(* CODESYS project Project1.project

Project tree, tasks and I/O mapping:
  PLC_AC500_V3 : PM5650-2ETH, ABB Automation Products GmbH, order no. 1SAPx41000R0278, version 3.4.1.0
    application Application
      task Task (cyclic, interval t#10ms, priority 15, watchdog t#20ms x 1) calls PLC_PRG
      CheckConfigurationObject
      program PLC_PRG [ST]
      data type motorIn
      data type motorOut
      data type fanIn
      data type fanOut
      data type valveIn
      data type valveOut
      function block AnalogSensor [ST]
      function block Valve [ST]: close, open, error
      function block AnalogValve [ST]
      function block Motor [ST]: start, stop, error, Init
      interface ILogging: Imethod1, Imethod2
      function block AbsLogging [ST]: Method1
      function block Compressor [ST]
      function block Condensor [ST]
      function block Evaporator [ST]
      function block Fan [ST]
      function block Pressure [ST]: Prop1, Prop2
      function block Temperature [ST]: HiAlarm, LoAlarm
      Diagnosis/
        text list Diag_IO_Bus
        text list Diag_V3_PLC
    IO_Bus : I/O-Bus, ABB Automation Products GmbH, version 3.4.0.0
    Interfaces : Interfaces, ABB Automation Products GmbH, version 3.4.1.0
      COM
      CAN
      Ethernet : Ethernet, ABB Automation Products GmbH, version 3.4.1.0
        ETH1 : IP Settings, ABB Automation Products GmbH, version 3.4.1.0
          NetConfig : NetConfig, ABB Automation Products GmbH, version 3.4.0.0
        ETH2 : IP Settings, ABB Automation Products GmbH, version 3.4.1.0
          NetConfig_1 : NetConfig, ABB Automation Products GmbH, version 3.4.0.0
        Protocols : Client Protocols, ABB Automation Products GmbH, version 3.4.1.0
    Extension_Bus : Extension Bus, ABB Automation Products GmbH, version 3.4.0.0
      Slot_1
      Slot_2
  Panel_CP600 : CP600 Control Panel, ABB Automation Products GmbH, order no. 1SAP500900R0001, version 2.10.0.0
    Panel Project
  libraries: VisuSymbols, 3.5.10.0 (System)
  text list GlobalTextList
*)

// PLC_AC500_V3/Application/motorIn
TYPE motorIn :
STRUCT
	StartMotor:BOOL;
	StopMotor:BOOL;
	Running:BOOL;
	Simulation:BOOL;
END_STRUCT
END_TYPE

// PLC_AC500_V3/Application/motorOut
TYPE motorOut :
STRUCT
	Output:BOOL;
	Error:BOOL;
END_STRUCT
END_TYPE

// PLC_AC500_V3/Application/fanIn
TYPE fanIn EXTENDS motorIn :
STRUCT
	fanSpeed:REAL;
END_STRUCT
END_TYPE

// PLC_AC500_V3/Application/fanOut
TYPE fanOut EXTENDS motorOut :
STRUCT
	outSpeed:REAL;
END_STRUCT
END_TYPE

// PLC_AC500_V3/Application/valveIn
TYPE valveIn :
STRUCT
	OpenCmd:BOOL;
	CloseCmd:BOOL;
	Opened:BOOL;
	Closed:BOOL;
END_STRUCT
END_TYPE

// PLC_AC500_V3/Application/valveOut
TYPE valveOut :
STRUCT
	Output:BOOL;
	Stall:BOOL;
END_STRUCT
END_TYPE

// PLC_AC500_V3/Application/AbsLogging/AMethod1
METHOD PUBLIC ABSTRACT AMethod1 : BOOL
VAR_INPUT
END_VAR

// PLC_AC500_V3/Application/AbsLogging/AMethod2
METHOD PUBLIC ABSTRACT AMethod2 : BOOL
VAR_INPUT
END_VAR

// PLC_AC500_V3/Application/PLC_PRG
PROGRAM PLC_PRG
VAR
	Compressor1:Compressor;
	Evaporator1:Evaporator;
	Condensor1:Condensor;
	
	TT1:Temperature; // Compressor Inlet Temperature / Evaporator Outlet Temperature
	TT2:Temperature; // Compressor Outlet Temperature / Condensor Inlet Temperature
	TT3:Temperature; // Condensor Outlet Temperature / Evaporator Inlet Temperature
	
	PT1:Pressure; // Compressor Inlet Pressure / Evaporator Outlet Pressure
	PT2:Pressure; // Compressor Outlet Pressure / Condensor Inlet Pressure
	PT3:Pressure; // Condensor Outlet Pressure / Evaporator Inlet Pressure
	PT4:Pressure; // 
	
	EEV1:AnalogValve; // Temperature Controlling Valve

	defrostTemperature:REAL;
	chillTemperature:REAL;
	Defrost:BOOL;
	Chilling:BOOL;
	
	var1:REAL;
END_VAR

Compressor1();
Condensor1();
Evaporator1();
PT1();
PT2();
PT3();
PT4();
TT1();
TT2();
TT3();
EEV1();
TT1.EngMax:=100;
TT1.EngMin:=0;
TT1.RawMax:=20000;
TT1.RawMin:=0;
TT1.Simulation:=TRUE;

TT2.EngMax:=100;
TT2.EngMin:=0;
TT2.RawMax:=20000;
TT2.RawMin:=0;
TT2.Simulation:=TRUE;

TT3.EngMax:=100;
TT3.EngMin:=0;
TT3.RawMax:=20000;
TT3.RawMin:=0;
TT3.Simulation:=TRUE;

PT1.EngMax:=10;
PT1.EngMin:=0;
PT1.RawMax:=20000;
PT1.RawMin:=0;
PT1.Simulation:=TRUE;

PT2.EngMax:=10;
PT2.EngMin:=0;
PT2.RawMax:=20000;
PT2.RawMin:=0;
PT2.Simulation:=TRUE;

PT3.EngMax:=10;
PT3.EngMin:=0;
PT3.RawMax:=20000;
PT3.RawMin:=0;
PT3.Simulation:=TRUE;

PT4.EngMax:=10;
PT4.EngMin:=0;
PT4.RawMax:=20000;
PT4.RawMin:=0;
PT4.Simulation:=TRUE;

PT1.Prop1:=10000;

var1:=PT1.Prop1;



Compressor1.Inputs.Simulation:=TRUE;
Condensor1.Inputs.Simulation:=TRUE;
Evaporator1.Inputs.Simulation:=TRUE;

// Code Section for Simulation & Testing

IF (Chilling) THEN
	Defrost:=FALSE;
	Condensor1.Inputs.StartMotor:=TRUE;
	Evaporator1.Inputs.StartMotor:=TRUE;
	EEV1.Inputs.OpenCmd:=TRUE;
	IF (TT1.PV > chillTemperature) THEN
		Compressor1.Inputs.StartMotor:=TRUE;
    ELSE
		Compressor1.Inputs.StopMotor:=TRUE;
	END_IF
ELSIF (NOT Chilling) AND (NOT Defrost) THEN
	Compressor1.Inputs.StopMotor:=TRUE;
	Condensor1.Inputs.StopMotor:=TRUE;
	Evaporator1.Inputs.StopMotor:=TRUE;
	EEV1.Inputs.CloseCmd:=TRUE;
END_IF


IF (Defrost) THEN
	Chilling:=FALSE;
	Compressor1.MotorSpeed:=0;
	Condensor1.Inputs.StartMotor:=TRUE;
	Evaporator1.Inputs.StartMotor:=TRUE;
	EEV1.Inputs.OpenCmd:=TRUE;
	IF ( TT1.PV < defrostTemperature) THEN
		Evaporator1.Inputs.fanSpeed:=100;
		EEV1.percentOpen:=10;
	ELSE
		Evaporator1.Inputs.fanSpeed:=0;
		EEV1.percentOpen:=0;
		Defrost:=FALSE;
	END_IF
ELSIF (NOT Chilling) AND (NOT Defrost) THEN
	Condensor1.Inputs.StopMotor:=TRUE;
	Evaporator1.Inputs.StopMotor:=TRUE;
	EEV1.Inputs.CloseCmd:=TRUE;
END_IF

IF (Chilling) AND (TT2.PV >= 60 AND TT2.PV <= 80 ) THEN
	Condensor1.Inputs.fanSpeed:=100;
ELSIF (Chilling) AND (TT2.PV >= 40 AND TT2.PV <= 60 ) THEN
	Condensor1.Inputs.fanSpeed:=75;
ELSIF (Chilling) AND (TT2.PV >= 20 AND TT2.PV <= 40  ) THEN
	Condensor1.Inputs.fanSpeed:=50;
ELSIF (Chilling) AND (TT2.PV >= 10 AND TT2.PV <= 20  ) THEN
	Condensor1.Inputs.fanSpeed:=25;
END_IF

IF (Chilling) AND ((TT1.PV - chillTemperature) >= 10 ) THEN
	Evaporator1.Inputs.fanSpeed:=100;
	IF (NOT defrost) AND (Chilling) THEN
		Compressor1.MotorSpeed:=100;
	END_IF	
	EEV1.percentOpen:=100;
ELSIF (Chilling) AND ((TT1.PV - chillTemperature) >= 8 ) THEN
	Evaporator1.Inputs.fanSpeed:=75;
	IF (NOT defrost) AND (Chilling) THEN
		Compressor1.MotorSpeed:=75;
	END_IF
	EEV1.percentOpen:=50;
ELSIF (Chilling) AND ((TT1.PV - chillTemperature) >= 6 ) THEN
	Evaporator1.Inputs.fanSpeed:=50;
	IF (NOT defrost) AND (Chilling) THEN
		Compressor1.MotorSpeed:=50;
	END_IF
	EEV1.percentOpen:=25;
ELSIF (Chilling) AND ((TT1.PV - chillTemperature) >= 4 ) THEN
	Evaporator1.Inputs.fanSpeed:=25;
	IF (NOT defrost) AND (Chilling) THEN
		Compressor1.MotorSpeed:=25;
	END_IF
	EEV1.percentOpen:=25;
ELSIF (Chilling) AND ((TT1.PV - chillTemperature) >= 2 ) THEN
	Evaporator1.Inputs.fanSpeed:=10;
	IF (NOT defrost) AND (Chilling) THEN
		Compressor1.MotorSpeed:=10;
	END_IF
	EEV1.percentOpen:=10;
END_IF

IF (Chilling) THEN
	IF (Compressor1.MotorSpeed <=100 AND Compressor1.MotorSpeed >=80) THEN
	PT1.SimIn:=50;
ELSIF (Compressor1.MotorSpeed <=80 AND Compressor1.MotorSpeed >=60) THEN
	PT1.SimIn:=45;
ELSIF (Compressor1.MotorSpeed <=60 AND Compressor1.MotorSpeed >=40) THEN
	PT1.SimIn:=30;
ELSIF (Compressor1.MotorSpeed <=40 AND Compressor1.MotorSpeed >=20) THEN
	PT1.SimIn:=25;
ELSIF (Compressor1.MotorSpeed =0) THEN
	PT1.SimIn:=20;
END_IF

IF (Condensor1.Inputs.fanSpeed <=100 AND Condensor1.Inputs.fanSpeed >=80) THEN
	PT2.SimIn:=12;
ELSIF (Condensor1.Inputs.fanSpeed <=80 AND Condensor1.Inputs.fanSpeed >=60) THEN
	PT2.SimIn:=14;
ELSIF (Condensor1.Inputs.fanSpeed <=60 AND Condensor1.Inputs.fanSpeed >=40) THEN
	PT2.SimIn:=16;
ELSIF (Condensor1.Inputs.fanSpeed <=40 AND Condensor1.Inputs.fanSpeed >=20) THEN
	PT2.SimIn:=18;
ELSIF (Condensor1.Inputs.fanSpeed =0) THEN
	PT2.SimIn:=20;
END_IF

IF (EEV1.percentOpen <=100 AND EEV1.percentOpen >=80) THEN
	PT3.SimIn:=5;
ELSIF (EEV1.percentOpen <=80 AND EEV1.percentOpen >=60) THEN
	PT3.SimIn:=7;
ELSIF (EEV1.percentOpen <=60 AND EEV1.percentOpen >=40) THEN
	PT3.SimIn:=9;
ELSIF (EEV1.percentOpen <=40 AND EEV1.percentOpen >=20) THEN
	PT3.SimIn:=11;
ELSIF (EEV1.percentOpen =0) THEN
	PT3.SimIn:=12;
END_IF

IF (Evaporator1.Inputs.fanSpeed <=100 AND Evaporator1.Inputs.fanSpeed >=80) THEN
	PT4.SimIn:=1;
ELSIF (Evaporator1.Inputs.fanSpeed <=80 AND Evaporator1.Inputs.fanSpeed >=60) THEN
	PT4.SimIn:=2;
ELSIF (Evaporator1.Inputs.fanSpeed <=60 AND Evaporator1.Inputs.fanSpeed >=40) THEN
	PT4.SimIn:=3;
ELSIF (Evaporator1.Inputs.fanSpeed <=40 AND Evaporator1.Inputs.fanSpeed >=20) THEN
	PT4.SimIn:=4;
ELSIF (Evaporator1.Inputs.fanSpeed =0) THEN
	PT4.SimIn:=5;
END_IF

END_IF

END_PROGRAM

// PLC_AC500_V3/Application/Compressor
FUNCTION_BLOCK Compressor EXTENDS Motor
VAR_INPUT
	MotorSpeed:REAL;
	InletPressure:REAL;
	InletTemperature:REAL;
	OutletPressure:REAL;
	OutletTemperature:REAL;
END_VAR
VAR_OUTPUT
	CompressorOn:BOOL;
	CompressorError:BOOL;
	CompressorSpeed:REAL;
END_VAR
VAR
END_VAR

SUPER^();

CompressorSpeed:=MotorSpeed;

END_FUNCTION_BLOCK

// PLC_AC500_V3/Application/Motor
FUNCTION_BLOCK PUBLIC Motor
VAR_INPUT
	Inputs:motorIn;
END_VAR
VAR_OUTPUT
	Outputs:motorOut;
END_VAR
VAR
	errorTimer:TON;
END_VAR

errorTimer(PT:=T#40S);
IF (Outputs.Output) AND (NOT Inputs.Running) AND (NOT Inputs.Simulation) THEN
		errorTimer.IN:=TRUE;
     IF (errorTimer.Q) THEN
         error();
		 errorTimer.IN:=FALSE;
     END_IF;
ELSIF (NOT Outputs.Output) AND (Inputs.Running) AND (NOT Inputs.Simulation) THEN
      errorTimer.IN:=TRUE;
     IF (errorTimer.Q) THEN
         error();
		 errorTimer.IN:=FALSE;
     END_IF;	
ELSE
         errorTimer.IN:=FALSE;
END_IF

IF(Inputs.StartMotor) THEN
	start();
END_IF

IF(Inputs.StopMotor) THEN
	stop();
END_IF

METHOD PROTECTED start : BOOL
VAR_INPUT
END_VAR
IF(Inputs.StartMotor) AND (NOT Outputs.Error) THEN
	Outputs.Output:=TRUE;
	Inputs.StartMotor:=FALSE;
END_IF
END_METHOD

METHOD PROTECTED stop : BOOL
VAR_INPUT
END_VAR
IF(Inputs.StopMotor) THEN
	Outputs.Output:=FALSE;
	Inputs.StopMotor:=FALSE;
END_IF
END_METHOD

METHOD PROTECTED error : BOOL
VAR_INPUT
END_VAR

VAR
	
END_VAR
IF (Outputs.Output) AND (Inputs.Running) AND (NOT Inputs.Simulation) THEN
		Outputs.Error:=TRUE;
	    Outputs.Output:=FALSE;	
ELSE
	Outputs.Error:=FALSE;
	errorTimer.IN:=FALSE;
END_IF
END_METHOD

METHOD PUBLIC Init : BOOL
VAR_INPUT
END_VAR
END_METHOD

END_FUNCTION_BLOCK

// PLC_AC500_V3/Application/Evaporator
FUNCTION_BLOCK Evaporator EXTENDS Fan
VAR_INPUT
	FanSpeed:REAL;
	InletPressure:REAL;
	InletTemperature:REAL;
	OutletPressure:REAL;
	OutletTemperature:REAL;
END_VAR
VAR_OUTPUT
	EvaporatorOn:BOOL;
	EvaporatorError:BOOL;
END_VAR
VAR
END_VAR

SUPER^();

END_FUNCTION_BLOCK

// PLC_AC500_V3/Application/Fan
FUNCTION_BLOCK Fan
VAR_INPUT
	Inputs:fanIn;
END_VAR
VAR_OUTPUT
	Outputs:fanOut;
END_VAR
VAR
	errorTimer:TON;
END_VAR

errorTimer(PT:=T#40S);
IF(Inputs.StartMotor) AND (NOT Outputs.Error) THEN
	Outputs.Output:=TRUE;
	WHILE(Outputs.outSpeed<Inputs.fanSpeed) DO
		Outputs.outSpeed:=Outputs.outSpeed+0.0001;
	END_WHILE
	Inputs.StartMotor:=FALSE;
END_IF


IF(Inputs.StopMotor) THEN
	Outputs.Output:=FALSE;
	WHILE(Outputs.outSpeed>0) DO
		Outputs.outSpeed:=Outputs.outSpeed-0.0001;
	END_WHILE
	Inputs.StopMotor:=FALSE;
END_IF


errorTimer(PT:=T#40S);
IF (Outputs.Output) AND (NOT Inputs.Running) AND (NOT Inputs.Simulation) THEN
     errorTimer.IN:=TRUE;
     IF (errorTimer.Q) THEN
         IF (Outputs.Output) AND (Inputs.Running) AND (NOT Inputs.Simulation) THEN
		     Outputs.Error:=TRUE;
	         Outputs.Output:=FALSE;	
         ELSE
	         Outputs.Error:=FALSE;
	         errorTimer.IN:=FALSE;
         END_IF
		 errorTimer.IN:=FALSE;
     END_IF;	
ELSIF (NOT Outputs.Output) AND (Inputs.Running) AND (NOT Inputs.Simulation) THEN
     errorTimer.IN:=TRUE;
     IF (errorTimer.Q) THEN
         IF (Outputs.Output) AND (Inputs.Running) AND (NOT Inputs.Simulation) THEN
		     Outputs.Error:=TRUE;
	         Outputs.Output:=FALSE;	
         ELSE
	         Outputs.Error:=FALSE;
	         errorTimer.IN:=FALSE;
         END_IF
		 errorTimer.IN:=FALSE;
     END_IF;	
ELSE
         errorTimer.IN:=FALSE;
END_IF

END_FUNCTION_BLOCK

// PLC_AC500_V3/Application/Condensor
FUNCTION_BLOCK Condensor EXTENDS Fan
VAR_INPUT
	FanSpeed:REAL;
	InletPressure:REAL;
	InletTemperature:REAL;
	OutletPressure:REAL;
	OutletTemperature:REAL;
END_VAR
VAR_OUTPUT
	CompressorOn:BOOL;
	CompressorError:BOOL;
END_VAR
VAR
END_VAR

SUPER^();

END_FUNCTION_BLOCK

// PLC_AC500_V3/Application/Temperature
FUNCTION_BLOCK Temperature EXTENDS AnalogSensor
VAR_INPUT
END_VAR
VAR_OUTPUT
	HiTempAlarm:BOOL;
	LoTempAlarm:BOOL;
END_VAR
VAR
END_VAR

SUPER^();
IF (PV<EngMin) THEN
	LoAlarm();
END_IF

IF (PV>EngMax) THEN
	HiAlarm();
END_IF

METHOD PUBLIC HiAlarm : BOOL
VAR_INPUT
END_VAR
IF (PV>EngMax) THEN
	HiTempAlarm:=TRUE;
ELSE
	HiTempAlarm:=FALSE;
END_IF
END_METHOD

METHOD LoAlarm : BOOL
VAR_INPUT
END_VAR
IF (PV<EngMin) THEN
	LoTempAlarm:=TRUE;
ELSE
	LoTempAlarm:=FALSE;
END_IF
END_METHOD

END_FUNCTION_BLOCK

// PLC_AC500_V3/Application/AnalogSensor
FUNCTION_BLOCK AnalogSensor
VAR_INPUT
	In:REAL;
	SimIn:REAL;
	RawMin:REAL;
	RawMax:REAL;
	EngMin:REAL;
	EngMax:REAL;
	Simulation:BOOL;
END_VAR
VAR_OUTPUT
	PV:REAL;
END_VAR
VAR
END_VAR

IF (Simulation) THEN
	PV:=SimIn;
ELSE
	PV:=((In-RawMin)*(EngMax-EngMin)/(RawMax-RawMin))+EngMin;
END_IF

END_FUNCTION_BLOCK

// PLC_AC500_V3/Application/Pressure
FUNCTION_BLOCK Pressure EXTENDS AnalogSensor
VAR_INPUT
END_VAR
VAR_OUTPUT 
	HiPresAlarm:BOOL;
	LoPresAlarm:BOOL;
END_VAR
VAR 
END_VAR

SUPER^();
IF (PV>EngMax) THEN
	HiPresAlarm:=TRUE;
ELSE
	HiPresAlarm:=FALSE;
END_IF


IF (PV<EngMin) THEN
	LoPresAlarm:=TRUE;
ELSE
	LoPresAlarm:=FALSE;
END_IF

PROPERTY PUBLIC Prop1 : REAL
SET
EngMax:=Prop1;
END_SET
GET
Prop1:=EngMax;
END_GET
END_PROPERTY

PROPERTY PUBLIC Prop2 : REAL
SET
END_SET
GET
END_GET
END_PROPERTY

END_FUNCTION_BLOCK

// PLC_AC500_V3/Application/AnalogValve
FUNCTION_BLOCK AnalogValve EXTENDS Valve
VAR_INPUT
	percentOpen:REAL;
END_VAR
VAR_OUTPUT
	outOpen:REAL;
END_VAR
VAR
END_VAR

SUPER^();
IF(Outputs.Output) THEN
	outOpen:=percentOpen;
ELSE
	outOpen:=0;
END_IF

END_FUNCTION_BLOCK

// PLC_AC500_V3/Application/Valve
FUNCTION_BLOCK Valve
VAR_INPUT
	Inputs:valveIn;
END_VAR
VAR_OUTPUT
	Outputs:valveOut;
END_VAR
VAR
	stallTimer:TON;
END_VAR

stallTimer(PT:=T#40S);

IF(Inputs.OpenCmd) THEN
	open();
END_IF

IF(Inputs.CloseCmd) THEN
	close();
END_IF

IF ((Inputs.OpenCmd) AND (NOT Inputs.Opened)) OR ((Inputs.CloseCmd) AND (NOT Inputs.Closed)) THEN
	stallTimer.IN:=TRUE;
	IF (stallTimer.Q) THEN
		error();
		stallTimer.IN:=FALSE;
	END_IF
ELSE
	stallTimer.IN:=FALSE;
END_IF

METHOD PRIVATE close : BOOL
VAR_INPUT
END_VAR
IF (Inputs.CloseCmd)  THEN
	Outputs.Output:=FALSE;
	Inputs.CloseCmd:=FALSE;
END_IF
END_METHOD

METHOD PRIVATE open : BOOL
VAR_INPUT
END_VAR
IF(Inputs.OpenCmd) AND (NOT Outputs.Stall) THEN
	Outputs.Output:=TRUE;
	Inputs.OpenCmd:=FALSE;
END_IF
END_METHOD

METHOD PRIVATE error : BOOL
VAR_INPUT
END_VAR
IF ((Inputs.OpenCmd) AND (NOT Inputs.Opened)) OR ((Inputs.CloseCmd) AND (NOT Inputs.Closed)) THEN
	Outputs.Stall:=TRUE;
ELSE
	Outputs.Stall:=FALSE;
END_IF
END_METHOD

END_FUNCTION_BLOCK

// PLC_AC500_V3/Application/ILogging
INTERFACE ILogging

METHOD Imethod1 : BOOL
VAR_INPUT
END_VAR
END_METHOD

METHOD Imethod2 : BOOL
VAR_INPUT
END_VAR
END_METHOD

END_INTERFACE

// PLC_AC500_V3/Application/AbsLogging
FUNCTION_BLOCK PUBLIC ABSTRACT AbsLogging
VAR_INPUT
END_VAR
VAR_OUTPUT
END_VAR
VAR
END_VAR

METHOD PUBLIC Method1 : BOOL
VAR_INPUT
END_VAR
END_METHOD

END_FUNCTION_BLOCK

(* text list Diag_IO_Bus (id | default | en)
  Err_1037 | Test error | Test error
  Err_12 | Test pulse error ->  Check wiring and sensor | Test pulse error ->  Check wiring and sensor
  Err_13 | Test pulse cross-talk error ->  Check wiring and sensor. If this error persists, replace I/O module. Contact ABB technical support. | Test pulse cross-talk error ->  Check wiring and sensor. If this error persists, replace I/O module. Contact ABB technical support.
  Err_16128 | Failed Max Wait Run | Failed Max Wait Run
  Err_16129 | Critical Error, see log | Critical Error, see log
  Err_16130 | Fatal Error, see log | Fatal Error, see log
  Err_16131 | Timeout -> Replace I/O module | Timeout -> Replace I/O module
  Err_16133 | Output data size mismatch | Output data size mismatch
  Err_16134 | Input data size mismatch | Input data size mismatch
  Err_16137 | Overflow diagnosis buffer -> Restart | Overflow diagnosis buffer -> Restart
  Err_16138 | Non-safety I/O: Voltage overflow on outputs (above UP3 level),  Safety I/O: Process voltage too high -> Check terminals/ check process voltage | Non-safety I/O: Voltage overflow on outputs (above UP3 level),  Safety I/O: Process voltage too high -> Check terminals/ check process voltage
  Err_16139 | Process voltage UP or UP3 too low -> Check process voltage | Process voltage UP or UP3 too low -> Check process voltage
  Err_16145 | Error setting parameters | Error setting parameters
  Err_16146 | Plausibility check failed (iParameter) ->  Check configuration | Plausibility check failed (iParameter) ->  Check configuration
  Err_16147 | Checksum error ->  Non-safety I/O: Replace I/O module. Safety I/O: Check safety configuration and CRCs for I- and F-Parameters. | Checksum error ->  Non-safety I/O: Replace I/O module. Safety I/O: Check safety configuration and CRCs for I- and F-Parameters.
  Err_16148 | PROFIsafe communication error ->  Restart I/O module. If this error persists, contact ABB technical support. | PROFIsafe communication error ->  Restart I/O module. If this error persists, contact ABB technical support.
  Err_16149 | No module data | No module data
  Err_16153 | PROFIsafe watchdog timed out ->  Restart I/O module. If this error persists, increase PROFIsafe watchdog time. | PROFIsafe watchdog timed out ->  Restart I/O module. If this error persists, increase PROFIsafe watchdog time.
  Err_16154 | Size of parameters excpeted by module differs from size provided by configuration ->  Check master or configuration | Size of parameters excpeted by module differs from size provided by configuration ->  Check master or configuration
  Err_16156 | F-Parameter configuration and address switch value do not match ->  Check I/O module F-Parameter configuration and module address switch value. | F-Parameter configuration and address switch value do not match ->  Check I/O module F-Parameter configuration and module address switch value.
  Err_16158 | Type of present module does not match configuration | Type of present module does not match configuration
  Err_16159 | Configured number of modules differs from found ones | Configured number of modules differs from found ones
  Err_16160 | At least one module failed during configuration | At least one module failed during configuration
  Err_16164 | Internal data exchange failure -> Replace I/O module | Internal data exchange failure -> Replace I/O module
  Err_16168 | Different hard-/firmware versions in the module -> Replace I/O module | Different hard-/firmware versions in the module -> Replace I/O module
  Err_16171 | Internal error ->  Replace I/O module | Internal error ->  Replace I/O module
  Err_16172 | Has not passed factory test | Has not passed factory test
  Err_16173 | No process voltage UP or UP3 -> Check process voltage | No process voltage UP or UP3 -> Check process voltage
  Err_16175 | Sensor voltage too low | Sensor voltage too low
  Err_16194 | Fatal error, not running any more | Fatal error, not running any more
  Err_16246 | Failed to start the parameterization of modules | Failed to start the parameterization of modules
  Err_16247 | Failed setting parameters | Failed setting parameters
  Err_16248 | Failed setting expected module | Failed setting expected module
  Err_16254 | Size of parameters excpeted by module differs from size provided by configuration | Size of parameters excpeted by module differs from size provided by configuration
  Err_18 | Test error | Test error
  Err_25 | Stuck-at error ->  Check I/O module wiring. Restart I/O module, if needed. If this error persists, replace I/O module. | Stuck-at error ->  Check I/O module wiring. Restart I/O module, if needed. If this error persists, replace I/O module.
  Err_257 | Wrong measurement, false temperature at the compensation channel | Wrong measurement, false temperature at the compensation channel
  Err_258 | AI531: Wrong measurement; potential difference is too high; CD522: PWM duty cycle out of duty area | AI531: Wrong measurement; potential difference is too high; CD522: PWM duty cycle out of duty area
  Err_260 | Measurement overflow ->  Check channel wiring and sensor power supply | Measurement overflow ->  Check channel wiring and sensor power supply
  Err_263 | Measurement underflow ->  Check channel wiring and sensor power supply | Measurement underflow ->  Check channel wiring and sensor power supply
  Err_266 | Short-circuit and cut wire or "out of range" | Short-circuit and cut wire or "out of range"
  Err_267 | Output/process voltage to small/low | Output/process voltage to small/low
  Err_273 | Test error | Test error
  Err_28 | Cross-talk error ->  Check I/O module wiring. Restart I/O module, if needed. If this error persists, replace I/O module. | Cross-talk error ->  Check I/O module wiring. Restart I/O module, if needed. If this error persists, replace I/O module.
  Err_3 | Discrepancy time expired ->  Check discrepancy time value, channel wiring and sensor. | Discrepancy time expired ->  Check discrepancy time value, channel wiring and sensor.
  Err_303 | Short-circuit at the analog input -> Check channel wiring | Short-circuit at the analog input -> Check channel wiring
  Err_304 | Analog value overflow or broken wire at an analog input -> Check value or check terminals | Analog value overflow or broken wire at an analog input -> Check value or check terminals
  Err_311 | Value difference too high ->  Adjust tolerance window for channels. Check channel wiring and sensor configuration. | Value difference too high ->  Adjust tolerance window for channels. Check channel wiring and sensor configuration.
  Err_524 | Stuck-at error | Stuck-at error
  Err_525 | Readback error ->  Check I/O module wiring. Restart I/O module, if needed. If this error persists, replace I/O module. | Readback error ->  Check I/O module wiring. Restart I/O module, if needed. If this error persists, replace I/O module.
  Err_530 | Class 3: Cross-talk error; Class 4: Internal fuse at 0V is defect. 0V not conected with GND. ->  Check I/O module wiring. Restart I/O module, if needed. If this error persists, replace I/O module. | Class 3: Cross-talk error; Class 4: Internal fuse at 0V is defect. 0V not conected with GND. ->  Check I/O module wiring. Restart I/O module, if needed. If this error persists, replace I/O module.
  Err_540 | Test error | Test error
  Err_555 | Internal error | Internal error
  Err_559 | Short-circuit at the digital output -> Check channel wiring | Short-circuit at the digital output -> Check channel wiring
  Err_775 | Measurement underflow at analog input ->  Check channel wiring | Measurement underflow at analog input ->  Check channel wiring
  Err_796 | Different configuration | Different configuration
  Err_8480 | Not supported protocol variant | Not supported protocol variant
  Err_8482 | Class 2: Timeout while initializing; Class 4: Timeout while waiting for ready status | Class 2: Timeout while initializing; Class 4: Timeout while waiting for ready status
  Err_8483 | Timeout during parameterization | Timeout during parameterization
  Err_8707 | PROFIsafe watchdog timed out | PROFIsafe watchdog timed out
  Err_8708 | Overvoltage | Overvoltage
  Err_8711 | Undervoltage | Undervoltage
  Err_8722 | Internal error | Internal error
  Err_8723 | Checksum error has occured in iParameters | Checksum error has occured in iParameters
  Err_8724 | PROFIsafe communication error | PROFIsafe communication error
  Err_8732 | Internal error  | Internal error 
  Err_8747 | Internal runtime error | Internal runtime error
  Err_8961 | Wrong parameter value, check configuration | Wrong parameter value, check configuration
  Err_8979 | Checksum error has occured in iParameter or F-Parameters | Checksum error has occured in iParameter or F-Parameters
  Err_8986 | Invalid configuration -> Check modules and parameterization | Invalid configuration -> Check modules and parameterization
  Err_8988 | F-Parameter configuration and address switch value do not match ->  Check I/O module F-Parameter configuration and module address switch value. | F-Parameter configuration and address switch value do not match ->  Check I/O module F-Parameter configuration and module address switch value.
  Err_9249 | Timeout while waiting for Reset | Timeout while waiting for Reset
  Err_9258 | Breakdown, communication lost | Breakdown, communication lost
  Err_9480 | I/O module removed from HotSwap terminal unit or defective module on HotSwap terminal unit -> Plug I/O module, replace I/O module | I/O module removed from HotSwap terminal unit or defective module on HotSwap terminal unit -> Plug I/O module, replace I/O module
  Err_9500 | Wrong I/O module plugged on HotSwap terminal unit -> Remove wrong I/O module and plug projected I/O module | Wrong I/O module plugged on HotSwap terminal unit -> Remove wrong I/O module and plug projected I/O module
  Err_9514 | No communication with I/O module on HotSwap terminal unit -> Replace I/O module | No communication with I/O module on HotSwap terminal unit -> Replace I/O module
  Err_9526 | I/O module does not support HotSwap functionality -> Power off system and replace I/O module | I/O module does not support HotSwap functionality -> Power off system and replace I/O module
  Err_9736 | HotSwap Terminal Unit required but not found | HotSwap Terminal Unit required but not found
  Err_9764 | Defective HotSwap Terminal Unit | Defective HotSwap Terminal Unit
  Err_9770 | No communication with HotSwap terminal unit -> Restart, if error persists replace terminal unit | No communication with HotSwap terminal unit -> Restart, if error persists replace terminal unit
  Hwd_14 | I/O-Bus | I/O-Bus
  Sub1_ | Module | Module
  Sub2_ | Channel | Channel *)

(* text list Diag_V3_PLC (id | default | en)
  Err_10 | Medium has almost used its complete spare capacity or is already dead, action required | Medium has almost used its complete spare capacity or is already dead, action required
  Err_17 | Error setting parameter | Error setting parameter
  Err_18 | At least one not found | At least one not found
  Err_19 | Unable to read at least one value | Unable to read at least one value
  Err_2 | Resource failure | Resource failure
  Err_20 | Invalid value of "Error LED" | Invalid value of "Error LED"
  Err_21 | Invalid value of "Check battery" | Invalid value of "Check battery"
  Err_22 | Error at initialization | Error at initialization
  Err_23 | Wrong version of firmware | Wrong version of firmware
  Err_24 | Invalid value of parameter "Diagnosis, stop on error class" | Invalid value of parameter "Diagnosis, stop on error class"
  Err_25 | Invalid value of parameter "Diagnosis, add Plc name to node name" | Invalid value of parameter "Diagnosis, add Plc name to node name"
  Err_26 | Invalid value of parameter "Reboot at powerfail" | Invalid value of parameter "Reboot at powerfail"
  Err_27 | Failed to set parameter "Reboot at powerfail" | Failed to set parameter "Reboot at powerfail"
  Err_28 | Value of parameter "Missed Cycle Task behaviour" is not in range | Value of parameter "Missed Cycle Task behaviour" is not in range
  Err_29 | Combination of plugged option boards is invalid | Combination of plugged option boards is invalid
  Err_3 | Timeout | Timeout
  Err_30 | Value of parameter "Priority Scheme" is not in range | Value of parameter "Priority Scheme" is not in range
  Err_8 | Empty or missing | Empty or missing
  Err_9 | Medium has used 80% of its spare capacity | Medium has used 80% of its spare capacity
  Hwd_0 | CPU | CPU
  Sub1_0 | CPU | CPU
  Sub1_14 | I/O-Bus | I/O-Bus
  Sub1_19 | Flashdisk | Flashdisk
  Sub1_21 | Display | Display
  Sub1_22 | Battery | Battery
  Sub2_0 | Device | Device
  Sub2_2 | Parameter | Parameter
  Sub2_5 | Index | Index
  Sub4_1 | too big | too big
  Sub4_2 | too small | too small
  Sub4_3 | unequal | unequal
  Sub4_4 | equal | equal *)
